(************************************************************************************************)
(*							Beckhoff Automation Poland											*)
(*								FB_ForceLockUnlock  v1.0										*)
(*									2.12.2010													*)
(*	Blok funkcyjny pozwalający w prosty sposób włączać i wyłączac hamulec silnika AMxxxx 		*)
(*							Potrzebna biblioteka MC2Drive 										*)
(*______________________________________________________________________________________________*)
FUNCTION_BLOCK FB_ForceLockUnlock
VAR_INPUT
	bForceLock : 		BOOL;
	bForceUnlock: 		BOOL;
END_VAR
VAR_OUTPUT
	bError: 			BOOL;
	bUnlocked: 			BOOL;
END_VAR
VAR_IN_OUT
	Axis: 				AXIS_REF;
END_VAR
VAR
	wWriteData:			WORD; 				(*1 - lock, 2 - unlock *)
	wReadData: 			WORD;
	ftWrite: 			F_TRIG;
	Delay1: 			TOF;
	fbSoEWrite: 		FB_SoEWrite;
	fbSoERead: 			FB_SoERead;
	wWriteDataOld: 		WORD;
END_VAR

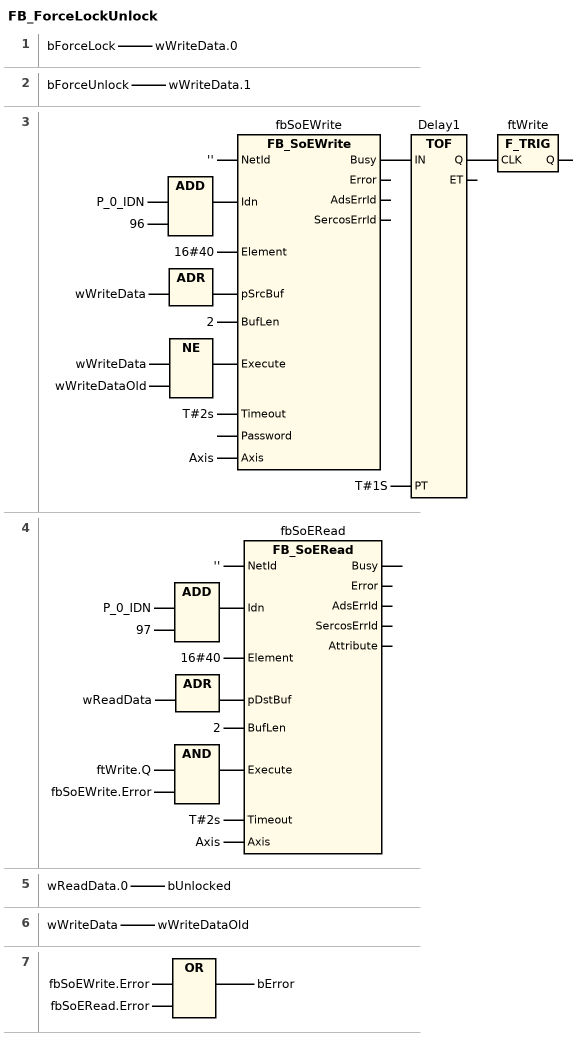
// NETWORK 1
wWriteData.0 := bForceLock;

// NETWORK 2
wWriteData.1 := bForceUnlock;

// NETWORK 3
fbSoEWrite(
    NetId := '',
    Idn := P_0_IDN + 96,
    Element := 16#40,
    pSrcBuf := ADR(wWriteData),
    BufLen := 2,
    Execute := wWriteData <> wWriteDataOld,
    Timeout := T#2s,
    Axis := Axis); // FB_SoEWrite
Delay1(IN := fbSoEWrite.Busy, PT := T#1S); // TOF
ftWrite(CLK := Delay1.Q); // F_TRIG

// NETWORK 4
fbSoERead(
    NetId := '',
    Idn := P_0_IDN + 97,
    Element := 16#40,
    pDstBuf := ADR(wReadData),
    BufLen := 2,
    Execute := ftWrite.Q AND fbSoEWrite.Error,
    Timeout := T#2s,
    Axis := Axis); // FB_SoERead

// NETWORK 5
bUnlocked := wReadData.0;

// NETWORK 6
wWriteDataOld := wWriteData;

// NETWORK 7
bError := fbSoEWrite.Error OR fbSoERead.Error;

END_FUNCTION_BLOCK

(* stored: Version 1.1.0.1, ProductVersion 3.1.4020.3
   POU FB_ForceLockUnlock: Id {3f888475-a708-4c26-9ed6-aa77d9805d0b}, SpecialFunc None *)
